DATA_BLOCK "PartDataManage_Part4_DB"
{ S7_Optimized_Access := 'TRUE' }
VERSION : 0.1
NON_RETAIN
"PartDataManage"

BEGIN

END_DATA_BLOCK

